// TIA Portal V19 export
DATA_BLOCK "SCALE_DB_TT"   // DB6
// stored: InstanceOfName SCALE, InstanceOfType FB
"SCALE"
   // VAR_INPUT
   //    "SCALE MIN" : Real;
   //    "SCALE MAX" : Real;
   //    INPUT : Int;
   //    RAW_MIN : Int;
   //    RAW_MAX : Int;
   // END_VAR
   // VAR_OUTPUT
   //    PV_VALUE : Real;
   // END_VAR
   // VAR_IN_OUT
   //    NORM_X : Real;
   // END_VAR
BEGIN
END_DATA_BLOCK
